// TIA Portal V17 export
// export: Created 2025-03-05T07:59:29.4310738Z, ExportSetting WithDefaults, DisplayName Totally Integrated Automation Portal, DisplayVersion V17 Update 8, DisplayName TIA Portal Openness, DisplayVersion V17 Update 8, DisplayName TIA Portal Version Control Interface, DisplayVersion V17, DisplayName SINAMICS Startdrive Advanced, DisplayVersion V17 SP2, DisplayName SINAMICS Startdrive G110M, G120, G120C, G120D, G120P, G115D, DisplayVersion V17 SP2, DisplayName SINAMICS Startdrive G130, G150, S120, S150, SINAMICS MV, S210, DisplayVersion V17 SP2, DisplayName STEP 7 Professional, DisplayVersion V17 Update 8, DisplayName SINUMERIK ONE STEP 7 Toolbox, DisplayVersion V17 Update 12, DisplayName SINUMERIK 840D sl STEP 7 Toolbox, DisplayVersion V17 Update 12, DisplayName STEP 7 Safety, DisplayVersion V17 Update 6, DisplayName WinCC Advanced, DisplayVersion V17 Update 8
FUNCTION_BLOCK "FB311_CHANNEL_PROGRAM_SELECTION"   // FB311, LAD
{ S7_Optimized_Access := 'FALSE' }
AUTHOR : ETXETAR
VERSION : 1.0
// stored: AutoNumber false, IsIECCheckEnabled false, SetENOAutomatically false, UDAEnableTagReadback false
   VAR_INPUT
      REQUEST : Bool;   // REQUEST
   END_VAR
   VAR_OUTPUT
      ALARM : Bool;
   END_VAR
   VAR_IN_OUT
      channelDB : "LBP_typeChanX";
   END_VAR
   VAR DB_SPECIFIC
      interlocksDB { S7_SetPoint := 'True'} : "CNC_PLC_INT_CH";
   END_VAR
   VAR
      FB7_INSTANCE { S7_SetPoint := 'True'} : "LBP_ReqPIService";
   END_VAR
   VAR_TEMP
      DB_NUMBER : DInt;   // DB NUMBER FOR ALARM AND HELP DECODING
      CHANNEL : Int;   // CHANNEL NUMBER MAX. NUMBER=10
   END_VAR
   VAR_TEMP   // added for the SCL form of the ladder/FBD networks
      _w1 : Bool;
      _w2 : Bool;
   END_VAR
BEGIN

NETWORK
TITLE = READ INSTANCE DB
      L     DINO;
      +     10#800000;
      T     #DB_NUMBER;
      L     DINO;
      L     10#310;
      -I;
      T     #CHANNEL;



REGION Network 2: RESET SELECTION
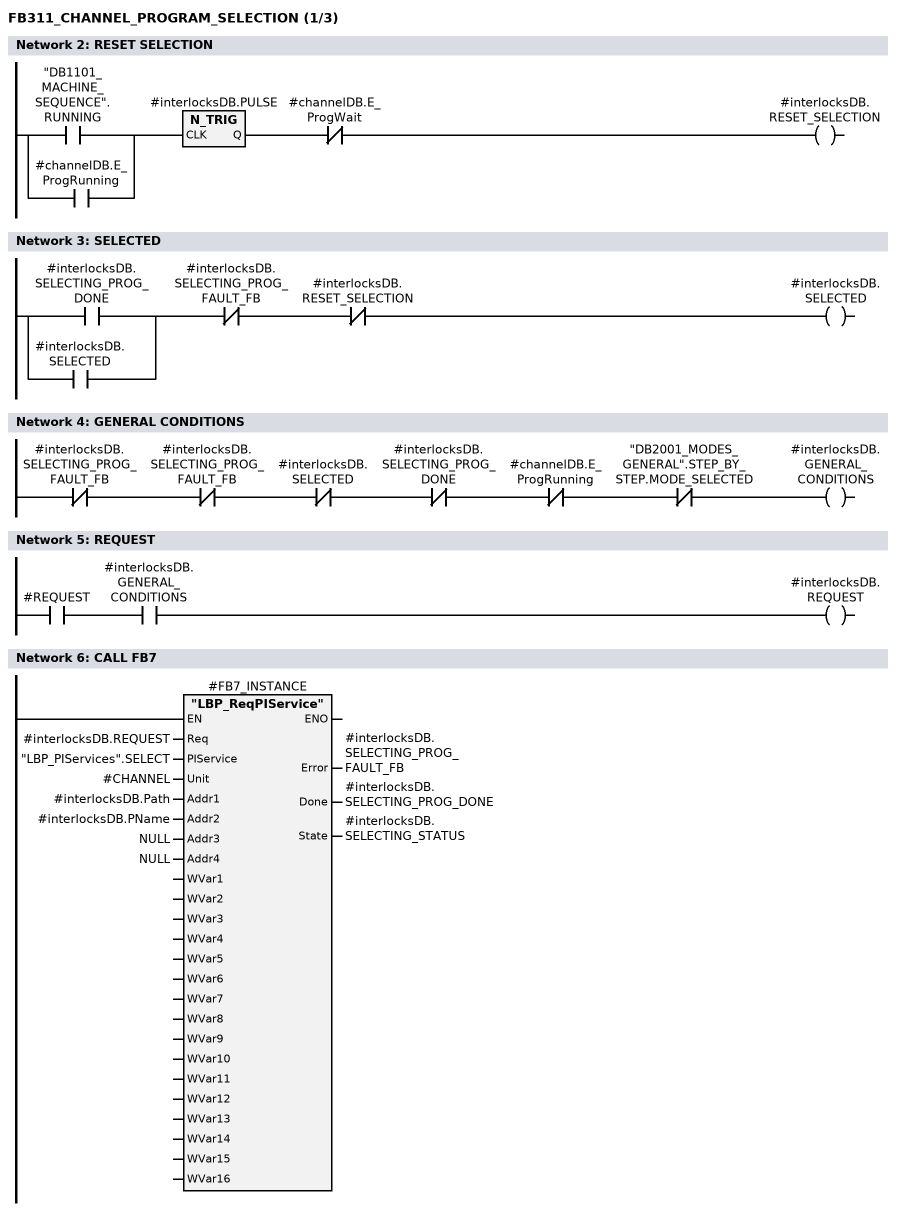
   RUNG wire#powerrail
      Contact( "DB1101_MACHINE_SEQUENCE".RUNNING )
      wire#w1
      N_Trig( #interlocksDB.PULSE )
      I_Contact( #channelDB.E_ProgWait )
      Coil( #interlocksDB.RESET_SELECTION )
   END_RUNG
   RUNG wire#powerrail
      Contact( #channelDB.E_ProgRunning )
   END_RUNG wire#w1
   // the same network as SCL:
   #_w1 := "DB1101_MACHINE_SEQUENCE".RUNNING OR #channelDB.E_ProgRunning;
   #_w2 := NOT #_w1 AND #interlocksDB.PULSE;   // falling edge
   #interlocksDB.PULSE := #_w1;
   #interlocksDB.RESET_SELECTION := #_w2 AND NOT #channelDB.E_ProgWait;
END_REGION

REGION Network 3: SELECTED
   RUNG wire#powerrail
      Contact( #interlocksDB.SELECTING_PROG_DONE )
      wire#w1
      I_Contact( #interlocksDB.SELECTING_PROG_FAULT_FB )
      I_Contact( #interlocksDB.RESET_SELECTION )
      Coil( #interlocksDB.SELECTED )
   END_RUNG
   RUNG wire#powerrail
      Contact( #interlocksDB.SELECTED )
   END_RUNG wire#w1
   // the same network as SCL:
   #interlocksDB.SELECTED := (#interlocksDB.SELECTING_PROG_DONE OR #interlocksDB.SELECTED) AND NOT #interlocksDB.SELECTING_PROG_FAULT_FB AND NOT #interlocksDB.RESET_SELECTION;
END_REGION

REGION Network 4: GENERAL CONDITIONS
   RUNG wire#powerrail
      I_Contact( #interlocksDB.SELECTING_PROG_FAULT_FB )
      I_Contact( #interlocksDB.SELECTING_PROG_FAULT_FB )
      I_Contact( #interlocksDB.SELECTED )
      I_Contact( #interlocksDB.SELECTING_PROG_DONE )
      I_Contact( #channelDB.E_ProgRunning )
      I_Contact( "DB2001_MODES_GENERAL".STEP_BY_STEP.MODE_SELECTED )
      Coil( #interlocksDB.GENERAL_CONDITIONS )
   END_RUNG
   // the same network as SCL:
   #interlocksDB.GENERAL_CONDITIONS := NOT #interlocksDB.SELECTING_PROG_FAULT_FB AND NOT #interlocksDB.SELECTING_PROG_FAULT_FB AND NOT #interlocksDB.SELECTED AND NOT #interlocksDB.SELECTING_PROG_DONE AND NOT #channelDB.E_ProgRunning AND NOT "DB2001_MODES_GENERAL".STEP_BY_STEP.MODE_SELECTED;
END_REGION

REGION Network 5: REQUEST
   RUNG wire#powerrail
      Contact( #REQUEST )
      Contact( #interlocksDB.GENERAL_CONDITIONS )
      Coil( #interlocksDB.REQUEST )
   END_RUNG
   // the same network as SCL:
   #interlocksDB.REQUEST := #REQUEST AND #interlocksDB.GENERAL_CONDITIONS;
END_REGION

REGION Network 6: CALL FB7
   RUNG wire#powerrail
      #FB7_INSTANCE(Req := #interlocksDB.REQUEST, PIService := "LBP_PIServices".SELECT, Unit := #CHANNEL, Addr1 := #interlocksDB.Path, Addr2 := #interlocksDB.PName, Addr3 := NULL, Addr4 := NULL, WVar1 :=, WVar2 :=, WVar3 :=, WVar4 :=, WVar5 :=, WVar6 :=, WVar7 :=, WVar8 :=, WVar9 :=, WVar10 :=, WVar11 :=, WVar12 :=, WVar13 :=, WVar14 :=, WVar15 :=, WVar16 :=, Error => #interlocksDB.SELECTING_PROG_FAULT_FB, Done => #interlocksDB.SELECTING_PROG_DONE, State => #interlocksDB.SELECTING_STATUS)
   END_RUNG
   // the same network as SCL:
   #FB7_INSTANCE(Req := #interlocksDB.REQUEST,   // "LBP_ReqPIService"
                 PIService := "LBP_PIServices".SELECT,
                 Unit := #CHANNEL,
                 Addr1 := #interlocksDB.Path,
                 Addr2 := #interlocksDB.PName,
                 Addr3 := NULL,
                 Addr4 := NULL,
                 Error => #interlocksDB.SELECTING_PROG_FAULT_FB,
                 Done => #interlocksDB.SELECTING_PROG_DONE,
                 State => #interlocksDB.SELECTING_STATUS);
END_REGION

REGION Network 7: PROGRAM SELECTION ALARM / FAULT
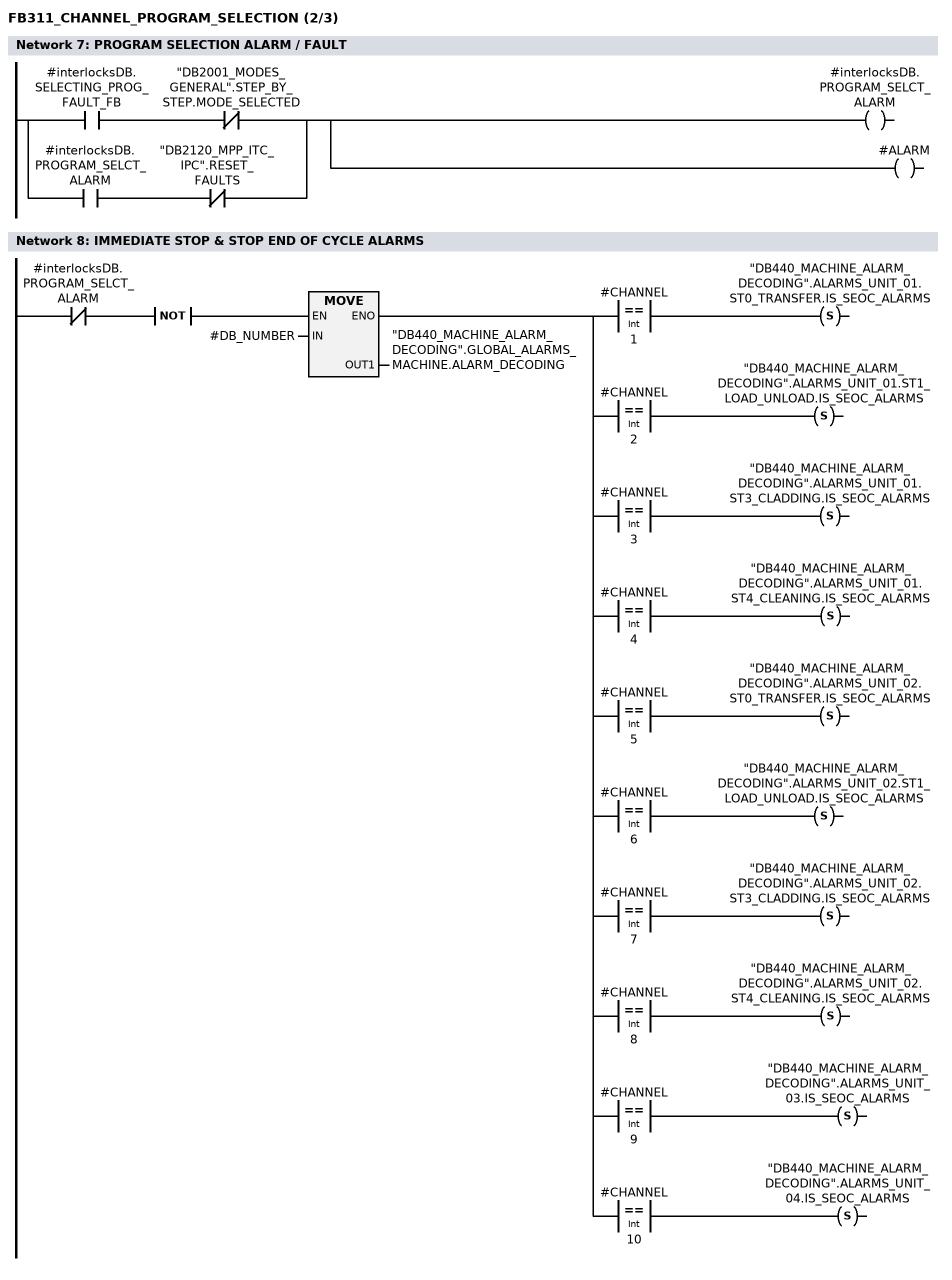
   RUNG wire#powerrail
      Contact( #interlocksDB.SELECTING_PROG_FAULT_FB )
      I_Contact( "DB2001_MODES_GENERAL".STEP_BY_STEP.MODE_SELECTED )
      wire#w1
      Coil( #interlocksDB.PROGRAM_SELCT_ALARM )
   END_RUNG
   RUNG wire#powerrail
      Contact( #interlocksDB.PROGRAM_SELCT_ALARM )
      I_Contact( "DB2120_MPP_ITC_IPC".RESET_FAULTS )
   END_RUNG wire#w1
   RUNG wire#w1
      Coil( #ALARM )
   END_RUNG
   // the same network as SCL:
   #interlocksDB.PROGRAM_SELCT_ALARM := (#interlocksDB.SELECTING_PROG_FAULT_FB AND NOT "DB2001_MODES_GENERAL".STEP_BY_STEP.MODE_SELECTED) OR (#interlocksDB.PROGRAM_SELCT_ALARM AND NOT "DB2120_MPP_ITC_IPC".RESET_FAULTS);
   #ALARM := #interlocksDB.PROGRAM_SELCT_ALARM;
END_REGION

REGION Network 8: IMMEDIATE STOP & STOP END OF CYCLE ALARMS
   RUNG wire#powerrail
      I_Contact( #interlocksDB.PROGRAM_SELCT_ALARM )
      Not()
      { S7_GenerateENO := "TRUE" } Move(in := #DB_NUMBER, out1 => "DB440_MACHINE_ALARM_DECODING".GLOBAL_ALARMS_MACHINE.ALARM_DECODING)
      wire#w1
      { S7_Templates := "SrcType := Int" } EQ_Contact(in1 := #CHANNEL, in2 := 1)
      S_Coil( "DB440_MACHINE_ALARM_DECODING".ALARMS_UNIT_01.ST0_TRANSFER.IS_SEOC_ALARMS )
   END_RUNG
   RUNG wire#w1
      { S7_Templates := "SrcType := Int" } EQ_Contact(in1 := #CHANNEL, in2 := 2)
      S_Coil( "DB440_MACHINE_ALARM_DECODING".ALARMS_UNIT_01.ST1_LOAD_UNLOAD.IS_SEOC_ALARMS )
   END_RUNG
   RUNG wire#w1
      { S7_Templates := "SrcType := Int" } EQ_Contact(in1 := #CHANNEL, in2 := 3)
      S_Coil( "DB440_MACHINE_ALARM_DECODING".ALARMS_UNIT_01.ST3_CLADDING.IS_SEOC_ALARMS )
   END_RUNG
   RUNG wire#w1
      { S7_Templates := "SrcType := Int" } EQ_Contact(in1 := #CHANNEL, in2 := 4)
      S_Coil( "DB440_MACHINE_ALARM_DECODING".ALARMS_UNIT_01.ST4_CLEANING.IS_SEOC_ALARMS )
   END_RUNG
   RUNG wire#w1
      { S7_Templates := "SrcType := Int" } EQ_Contact(in1 := #CHANNEL, in2 := 5)
      S_Coil( "DB440_MACHINE_ALARM_DECODING".ALARMS_UNIT_02.ST0_TRANSFER.IS_SEOC_ALARMS )
   END_RUNG
   RUNG wire#w1
      { S7_Templates := "SrcType := Int" } EQ_Contact(in1 := #CHANNEL, in2 := 6)
      S_Coil( "DB440_MACHINE_ALARM_DECODING".ALARMS_UNIT_02.ST1_LOAD_UNLOAD.IS_SEOC_ALARMS )
   END_RUNG
   RUNG wire#w1
      { S7_Templates := "SrcType := Int" } EQ_Contact(in1 := #CHANNEL, in2 := 7)
      S_Coil( "DB440_MACHINE_ALARM_DECODING".ALARMS_UNIT_02.ST3_CLADDING.IS_SEOC_ALARMS )
   END_RUNG
   RUNG wire#w1
      { S7_Templates := "SrcType := Int" } EQ_Contact(in1 := #CHANNEL, in2 := 8)
      S_Coil( "DB440_MACHINE_ALARM_DECODING".ALARMS_UNIT_02.ST4_CLEANING.IS_SEOC_ALARMS )
   END_RUNG
   RUNG wire#w1
      { S7_Templates := "SrcType := Int" } EQ_Contact(in1 := #CHANNEL, in2 := 9)
      S_Coil( "DB440_MACHINE_ALARM_DECODING".ALARMS_UNIT_03.IS_SEOC_ALARMS )
   END_RUNG
   RUNG wire#w1
      { S7_Templates := "SrcType := Int" } EQ_Contact(in1 := #CHANNEL, in2 := 10)
      S_Coil( "DB440_MACHINE_ALARM_DECODING".ALARMS_UNIT_04.IS_SEOC_ALARMS )
   END_RUNG
   // the same network as SCL:
   // ENO of a box is taken as its EN; it also drops when the box reports an error
   #_w1 := NOT (NOT #interlocksDB.PROGRAM_SELCT_ALARM);
   IF #_w1 THEN "DB440_MACHINE_ALARM_DECODING".GLOBAL_ALARMS_MACHINE.ALARM_DECODING := #DB_NUMBER; END_IF;
   IF #_w1 AND (#CHANNEL = 1) THEN
       "DB440_MACHINE_ALARM_DECODING".ALARMS_UNIT_01.ST0_TRANSFER.IS_SEOC_ALARMS := TRUE;
   END_IF;
   IF #_w1 AND (#CHANNEL = 2) THEN
       "DB440_MACHINE_ALARM_DECODING".ALARMS_UNIT_01.ST1_LOAD_UNLOAD.IS_SEOC_ALARMS := TRUE;
   END_IF;
   IF #_w1 AND (#CHANNEL = 3) THEN
       "DB440_MACHINE_ALARM_DECODING".ALARMS_UNIT_01.ST3_CLADDING.IS_SEOC_ALARMS := TRUE;
   END_IF;
   IF #_w1 AND (#CHANNEL = 4) THEN
       "DB440_MACHINE_ALARM_DECODING".ALARMS_UNIT_01.ST4_CLEANING.IS_SEOC_ALARMS := TRUE;
   END_IF;
   IF #_w1 AND (#CHANNEL = 5) THEN
       "DB440_MACHINE_ALARM_DECODING".ALARMS_UNIT_02.ST0_TRANSFER.IS_SEOC_ALARMS := TRUE;
   END_IF;
   IF #_w1 AND (#CHANNEL = 6) THEN
       "DB440_MACHINE_ALARM_DECODING".ALARMS_UNIT_02.ST1_LOAD_UNLOAD.IS_SEOC_ALARMS := TRUE;
   END_IF;
   IF #_w1 AND (#CHANNEL = 7) THEN
       "DB440_MACHINE_ALARM_DECODING".ALARMS_UNIT_02.ST3_CLADDING.IS_SEOC_ALARMS := TRUE;
   END_IF;
   IF #_w1 AND (#CHANNEL = 8) THEN
       "DB440_MACHINE_ALARM_DECODING".ALARMS_UNIT_02.ST4_CLEANING.IS_SEOC_ALARMS := TRUE;
   END_IF;
   IF #_w1 AND (#CHANNEL = 9) THEN
       "DB440_MACHINE_ALARM_DECODING".ALARMS_UNIT_03.IS_SEOC_ALARMS := TRUE;
   END_IF;
   IF #_w1 AND (#CHANNEL = 10) THEN
       "DB440_MACHINE_ALARM_DECODING".ALARMS_UNIT_04.IS_SEOC_ALARMS := TRUE;
   END_IF;
END_REGION

REGION Network 9: PROGRAMMING ALARM
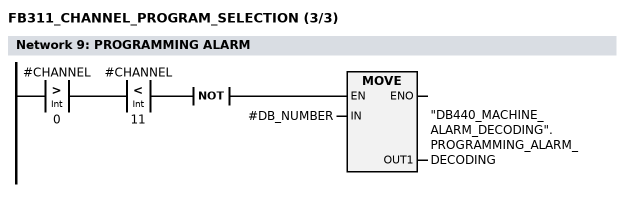
   RUNG wire#powerrail
      { S7_Templates := "SrcType := Int" } GT_Contact(in1 := #CHANNEL, in2 := 0)
      { S7_Templates := "SrcType := Int" } LT_Contact(in1 := #CHANNEL, in2 := 11)
      Not()
      Move(in := #DB_NUMBER, out1 => "DB440_MACHINE_ALARM_DECODING".PROGRAMMING_ALARM_DECODING)
   END_RUNG
   // the same network as SCL:
   IF NOT ((#CHANNEL > 0) AND (#CHANNEL < 11)) THEN
       "DB440_MACHINE_ALARM_DECODING".PROGRAMMING_ALARM_DECODING := #DB_NUMBER;
   END_IF;
END_REGION
END_FUNCTION_BLOCK
